Yaskawa INFORM job: TEST3.JBI

/JOB
//NAME TEST3
///FOLDERNAME INNE
//POS
///NPOS 4,4,4,0,0,0
///TOOL 0
///POSTYPE PULSE
///PULSE
C00000=72905,-45160,-22814,18302,91973,24343
C00001=-94322,46130,6191,-23852,113824,-36185
C00002=-191446,-39195,-66709,-21464,120818,-28385
C00003=-29931,41877,1808,23590,115288,35168
BC00000=167457,70930,653105
BC00001=167457,70930,350739
BC00002=167457,70930,350739
BC00003=167457,70930,350739
EC00000=0,0
EC00001=0,0
EC00002=0,556475
EC00003=0,556475
//INST
///DATE 2023/10/04 15:16
///ATTR SC,RW
///GROUP1 RB1,BS1
///GROUP2 ST1
NOP
'test3
MOVJ C00000 BC00000 VJ=100.00  +MOVJ EC00000 VJ=100.00
MOVJ C00001 BC00001 VJ=100.00  +MOVJ EC00001 VJ=100.00
MOVJ C00002 BC00002 VJ=100.00  +MOVJ EC00002 VJ=100.00
MOVJ C00003 BC00003 VJ=100.00  +MOVJ EC00003 VJ=100.00
END
